      FOR devIdx := groupBase TO groupBase + 3 DO
        IF devIdx <= 19 THEN
          IF GVL.Direction[devIdx] THEN
            reverseMode := TRUE;
          END_IF;
          IF GVL.Vin[devIdx] > 0 AND NOT GVL.CommFault[devIdx] AND NOT GVL.SafetyShutdown[devIdx] THEN
            activeInGroupX10 := activeInGroupX10 + 1;
          END_IF;
        END_IF;
      END_FOR;

      IF reverseMode THEN
        perDeviceLimitX10 := REAL_TO_UINT(GVL_Constant.BIC24_IOUT_MAX_REV * 10.0);
      ELSE
        perDeviceLimitX10 := REAL_TO_UINT(GVL_Constant.BIC24_IOUT_MAX_FWD * 10.0);
      END_IF;

      groupLimitFwdX10 := activeInGroupX10 * perDeviceLimitFwdX10;
      groupLimitRevX10 := activeInGroupX10 * perDeviceLimitRevX10;
      GVL.NumericOutput[112 + groupIdx] := SHL(TO_DWORD(groupLimitFwdX10), 16) OR TO_DWORD(groupLimitRevX10);
    END_FOR;

     (* DIAGNOSTIC: Group 3/4 isolation verification in valid slots [116..120].
       Note: some HMI links show only low 16-bit values from DWORD tags, so publish one value per slot.
       [116] raw Group3 Vout input  = NumericInput[GroupInputBase[2]]
       [117] raw Group4 Vout input  = NumericInput[GroupInputBase[3]]
       [118] applied Group3 VoutSetpoint (dev12, x100 engineering)
       [119] applied Group4 VoutSetpoint (dev16, x100 engineering)
       [120] absolute command delta = ABS(LastVoutSetpoint[12] - LastVoutSetpoint[16]); 0 means both groups are being commanded identically *)
     (* [116] LastVoutSetpoint[12]: last Vout CAN command sent to dev12 (Group3 first BIC) *)
     GVL.NumericOutput[116] := TO_DWORD(LastVoutSetpoint[12]);
     (* [117] LastVoutSetpoint[16]: last Vout CAN command sent to dev16 (Group4 first BIC) *)
     GVL.NumericOutput[117] := TO_DWORD(LastVoutSetpoint[16]);
     (* [118] Dev12 mode flags: bit0=Voltage, bit1=Current, bit2=OutputOn, bit3=OperationOn, bits 8-11 same for dev16 *)
     GVL.NumericOutput[118] := SHL(TO_DWORD(GVL.Voltage[12]), 0) OR
                                SHL(TO_DWORD(GVL.Current[12]), 1) OR
                                SHL(TO_DWORD(GVL.OutputOn[12]), 2) OR
                                SHL(TO_DWORD(GVL.OperationOn[12]), 3) OR
                                SHL(TO_DWORD(GVL.Voltage[16]), 8) OR
                                SHL(TO_DWORD(GVL.Current[16]), 9) OR
                                SHL(TO_DWORD(GVL.OutputOn[16]), 10) OR
                                SHL(TO_DWORD(GVL.OperationOn[16]), 11);
     (* [119] GroupMaster[2] (G3) and GroupMaster[3] (G4); -1 = no master assigned *)
     GVL.NumericOutput[119] := SHL(TO_DWORD(INT_TO_UINT(GVL.GroupMaster[2])), 16) OR TO_DWORD(INT_TO_UINT(GVL.GroupMaster[3]));
     (* [120] Raw NumericInput[GroupInputBase[2]] = Group3 Vout input; compare with [117] to check Morphee PDO *)
     GVL.NumericOutput[120] := TO_DWORD(GVL.NumericInput[GVL.GroupInputBase[3]]);
END_IF;
END_METHOD

END_FUNCTION_BLOCK

(* stored: Version 1.1.0.1, ProductVersion 3.1.4024.13
   POU EthercatManager: Id {f73e9df5-d22b-4027-8eaf-ab5cb0520b6c}, SpecialFunc None
   Method ApplyCommands: Id {ee2cc573-91f9-4349-9f7c-e0af36fc135f}
   Method ProcessInputs: Id {b2c3d4e5-2345-6789-0123-456789abcdef}
   Method ReadLimits: Id {0cee76ab-620c-4b89-985e-d5b10c795a48}
   Method UpdateOutputs: Id {c3d4e5f6-3456-7890-1234-56789abcdef0} *)
